Universal Robots PolyScope program: script_code_urp.urp

Program script_code_urp (installation=default directory=/programs createdIn=5.16.0 lastSavedIn=5.16.0 robotSerialNumber=20185000234)
Calibrated DH parameters: a=[-0.000035, -0.454311, -0.571382, -0.000018, 0.000029, 0]; d=[0.181274, 173.943413, -175.385997, 1.617009, 0.119839, 0.116075]; alpha=[1.570668, -0.002363, -0.002402, 1.570676, -1.571489, 0]; deltaTheta=[0, -0.735494, 0.741561, -0.006062, -0.000002, 0]
InitVariablesNode
Robot Program (runOnlyOnce=false)
  Script file /programs/script_code.script
    | socket_open("172.21.0.2", 8000, "abcd")
    | 
    | a = p[-1.421, -1.736, -2.43, -0.5, 1.606, 0]
    | movej(a, a=0.3, v=0.3)
    | 
    | b = p[-0.194, -0.6, 0.066, 2.61, -1.806, -0.019]
    | 
    | i = 0
    | while i < 5:
    |     sleep(2)
    |     i = i + 1
    | end
    | 
    | #movej(b, a=0.3, v=0.3)
  Halt
